# EPICS alarm handler configuration: mps_database/bareTest/alarms/areas/mpln_l3b_mp05.alhConfig
GROUP NULL MPLN:L3B:MP05:1
$ALIAS MPS Link Node 71
$GUIDANCE
LTUH MPS
   Group Name: MPLN:L3B:MP05:1
   Summary PV:  MPLN:L3B:MP05:1:STATSUMY
$END
CHANNEL  MPLN:L3B:MP05:1    MPLN:L3B:MP05:1:MPS_EN_RBV		-----
CHANNEL  MPLN:L3B:MP05:1    MPLN:L3B:MP05:1:LC1_MODE_RBV		-----
